(* IEC 61131-3 sources: programs/VI-54/VI-54_20171205/VI-54_20171205/Stations/Screen/LseClass170718/Class/EventJournal (part 2) *)

    // Koordinaten bestimmen
    tmpRoom.xy1.x += to_int(EventConfig.aColumnWidths[3]);
    tmpRoom.xy2.x += to_int(EventConfig.aColumnWidths[3]);

    Graphic.Line( x1      := tmpRoom.xy1.x,
                  y1      := tmpRoom.xy1.y,
                  x2      := tmpRoom.xy2.x,
                  y2      := tmpRoom.xy2.y,
                  attrib  := T_SOLID,
                  color   := sColor);

  end_if;

  //-----------------------------------------------------------------------------------------

END_FUNCTION

FUNCTION VIRTUAL EventJournal::GetEventText
	VAR_INPUT
		pEntry 	: ^_SINGLEALARM;
	END_VAR
	VAR_OUTPUT
		pEventTxt 	: ^_CHAR;
	END_VAR
  VAR
    pText       : ^_CHAR;
    tmpColor    : _COLOR;
    tmpIndex    : UINT;
   	MemVarLabel	: _MEM_VARLABEL;			// pointer to structure to get variables or constants
  END_VAR

  //===============================================================================================
  //  INIT
  //===============================================================================================
  pEventTxt := NIL;

  //===============================================================================================
  //  Übergabeparameter prüfen
  //===============================================================================================
  if (pEntry = NIL) then
    if (IsCon_coSystemLogging = True) then    // KaiAnd
      coSystemLogging.LogEventText("EventJournal::GetEventText(): Übergabeparameter pEntry = NIL" );
    end_if;
    return;
  end_if;

  //===============================================================================================
  //  create the memvarlabel for the defined text
  //===============================================================================================
 	init_MEM_VARLABEL(#MemVarLabel);

  if (pEntry^.ptr <> NIL) then
		// allocate the memory
    if ((Graphic.Memory(#MemVarLabel.ptr, sizeof(_VARLABEL))) <> NIL) then

      MemVarLabel.no := 1;
      MemVarLabel.ptr^.no := 1;
      MemVarLabel.ptr^.info[0].state := POINTER_CHAR;
      MemVarLabel.ptr^.info[0].value := pEntry^.ptr$DINT;
    end_if;
  end_if;

  //===============================================================================================
  //  UNTERSCHEIDUNG DER VERSCHIEDENEN EINTRÄGE
  //===============================================================================================
  case (pEntry^.entrytype) of

      //=======================================================================================
      //  Steuerung wurde eingeschaltet
      //---------------------------------------------------------------------------------------
      EVENT_SWITCHON:

        pEventTxt$^void := NewDoScheme(x0 := EventConfig.SystemOnOff.list,
                                      x1 := EVENT_TEXTSWITCHON,
                                      x2 := EventConfig.SystemOnOff.no);

        if (pEventTxt = NIL) then
          StrNCpy(p0:= #tmpEvTxt[0], x1:=sizeof(_CHAR), p2:="System on", x3:=1, ml:=sizeof(tmpEvTxt)/sizeof(_CHAR));
          pEventTxt := #tmpEvTxt[0];
        end_if;

      //=======================================================================================
      //  Steuerung wurde ausgeschaltet
      //---------------------------------------------------------------------------------------
      EVENT_SWITCHOFF:

        pEventTxt$^void := NewDoScheme(x0 := EventConfig.SystemOnOff.list,
                                      x1 := EVENT_TEXTSWITCHOFF,
                                      x2 := EventConfig.SystemOnOff.no);

        if (pEventTxt = NIL) then
          StrNCpy(p0:= #tmpEvTxt[0], x1:=sizeof(_CHAR), p2:="System off", x3:=1, ml:=sizeof(tmpEvTxt)/sizeof(_CHAR));
          pEventTxt := #tmpEvTxt[0];
        end_if;

      //=======================================================================================
      //  Betriebsart wurde umgeschaltet
      //---------------------------------------------------------------------------------------
      EVENT_OPCHANGE:

        // je nach Betriebsart anderen Text aus Liste holen
        case (pEntry^.para[2]$t_e_OPMode) of
          OPMode_Init:      tmpIndex := EVENT_TEXTOPMODEINIT;
          OPMode_Stop:      tmpIndex := EVENT_TEXTOPMODESTOP;
          OPMode_Setup:     tmpIndex := EVENT_TEXTOPMODESETUP;
          OPMode_Manual:    tmpIndex := EVENT_TEXTOPMODEMANUAL;
          OPMode_SemiAuto:  tmpIndex := EVENT_TEXTOPMODESEMIAUTO;
          OPMode_Automatic: tmpIndex := EVENT_TEXTOPMODEAUTOMATIC;
        else
          if (IsCon_coSystemLogging = True) then    // KaiAnd
            coSystemLogging.LogEventText("EventJournal::GetEventText(): unbekannter Betriebsmodus eingetragen" );
          end_if;
          tmpIndex := EVENT_TEXTOPMODEINIT;
        end_case;

        // Text aus Textliste holen
        pEventTxt$^void := NewDoScheme(x0 := EventConfig.OPMode.list,
                                       x1 := tmpIndex,
                                       x2 := EventConfig.OPMode.no);

        // Prüfen ob Text gefunden wurde
        if (pEventTxt = NIL) then
          StrNCpy(p0:= #tmpEvTxt[0], x1:=sizeof(_CHAR), p2:="change OP mode", x3:=1, ml:=sizeof(tmpEvTxt)/sizeof(_CHAR));
          pEventTxt := #tmpEvTxt[0];
        end_if;

      //=======================================================================================
      //  Login
      //---------------------------------------------------------------------------------------
      EVENT_USERLOGIN:

        pText := StupidTextScheme(Event_TextLogin, EventConfig.LoginLogout.no);
        pText := make_parameterstring(pText, #MemVarLabel, _TRUE);

        // Prüfen ob Text verfügbar
        if (pText = NIL) then
          StrNCpy(p0:= #tmpEvTxt[0], x1:=sizeof(_CHAR), p2:="user login text not found", x3:=1, ml:=sizeof(tmpEvTxt)/sizeof(_CHAR));
        else
          StrNCpy(p0:= #tmpEvTxt[0], x1:=sizeof(_CHAR), p2:=pText, x3:=sizeof(_CHAR), ml:=sizeof(tmpEvTxt)/sizeof(_CHAR));
        end_if;
        pEventTxt := #tmpEvTxt[0];

      //=======================================================================================
      //  Logout
      //---------------------------------------------------------------------------------------
      EVENT_USERLOGOUT:

        // Alarmtext bestimmen
        pText := StupidTextScheme(EVENT_TEXTLOGOUT, EventConfig.LoginLogout.no);
        pText := make_parameterstring(pText, #MemVarLabel, _TRUE);

        // Prüfen ob Text verfügbar
        if (pText = NIL) then
          StrNCpy(p0:= #tmpEvTxt[0], x1:=sizeof(_CHAR), p2:="user logout text not found", x3:=1, ml:=sizeof(tmpEvTxt)/sizeof(_CHAR));
        else
          StrNCpy(p0:= #tmpEvTxt[0], x1:=sizeof(_CHAR), p2:=pText, x3:=sizeof(_CHAR), ml:=sizeof(tmpEvTxt)/sizeof(_CHAR));
        end_if;
        pEventTxt := #tmpEvTxt[0];

      //=======================================================================================
      //  Benutzer-Event
      //---------------------------------------------------------------------------------------
      EVENT_USEREVENT:

        pEventTxt$^void := pEntry^.ptr;

      //=======================================================================================
      //  Datumsänderung
      //---------------------------------------------------------------------------------------
      EVENT_DATECHANGE:

        pEventTxt := GetTextEventDateChange(pEntry);

      //=======================================================================================
      //  Zeitänderung
      //---------------------------------------------------------------------------------------
      EVENT_TIMECHANGE:

        pEventTxt := GetTextEventTimeChange(pEntry);

      //=======================================================================================
      //  Wertänderung
      //---------------------------------------------------------------------------------------
      EVENT_VALUECHANGE:

        pEventTxt := GetTextEventValueChange(pEntry);

      //=======================================================================================
      //  Menüeintrags-Änderung
      //---------------------------------------------------------------------------------------
      EVENT_MENUCHANGE:

        pEventTxt := GetTextEventMenueChange(pEntry);

      //=======================================================================================
      //  Alarm
      //---------------------------------------------------------------------------------------
      EVENT_ALARM :
        // Alarmtext bestimmen
        pEventTxt := create_alarmtext(p0:= pEntry, x1:=false, p2:=#tmpColor);

        // Prüfen ob Text verfügbar
        if (pEventTxt = NIL) then
          if (IsCon_coSystemLogging = True) then    // KaiAnd
            coSystemLogging.LogEventText("EventJournal::GetEventText(): Text für den Alarm nicht gefunden" );
          end_if;
        end_if;

      //=======================================================================================
      //  System Meldungen Kategorie 1
      //---------------------------------------------------------------------------------------
      Event_SystemCat1 :

        // Alarmtext bestimmen
        pText := StupidTextScheme(pEntry^.para[2], EventConfig.SystemEntryCategory1.no);
        pText := make_parameterstring(pText, #MemVarLabel, _TRUE);

        // Prüfen ob Text verfügbar
        if (pText = NIL) then
          StrNCpy(p0:= #tmpEvTxt[0], x1:=sizeof(_CHAR), p2:="system text cat1 not found", x3:=1, ml:=sizeof(tmpEvTxt)/sizeof(_CHAR));
        else
          StrNCpy(p0:= #tmpEvTxt[0], x1:=sizeof(_CHAR), p2:=pText, x3:=sizeof(_CHAR), ml:=sizeof(tmpEvTxt)/sizeof(_CHAR));
        end_if;
        pEventTxt := #tmpEvTxt[0];

      //=======================================================================================
      //  System Meldungen Kategorie 2
      //---------------------------------------------------------------------------------------
      Event_SystemCat2 :

        // Alarmtext bestimmen
        pText := StupidTextScheme(pEntry^.para[2], EventConfig.SystemEntryCategory2.no);
        pText := make_parameterstring(pText, #MemVarLabel, _TRUE);

        // Prüfen ob Text verfügbar
        if (pText = NIL) then
          StrNCpy(p0:= #tmpEvTxt[0], x1:=sizeof(_CHAR), p2:="system text cat2 not found", x3:=1, ml:=sizeof(tmpEvTxt)/sizeof(_CHAR));
        else
          StrNCpy(p0:= #tmpEvTxt[0], x1:=sizeof(_CHAR), p2:=pText, x3:=sizeof(_CHAR), ml:=sizeof(tmpEvTxt)/sizeof(_CHAR));
        end_if;
        pEventTxt := #tmpEvTxt[0];

      //=======================================================================================
      //  System Meldungen Kategorie 3
      //---------------------------------------------------------------------------------------
      Event_SystemCat3 :

        // Alarmtext bestimmen
        pText := StupidTextScheme(pEntry^.para[2], EventConfig.SystemEntryCategory3.no);
        pText := make_parameterstring(pText, #MemVarLabel, _TRUE);

        // Prüfen ob Text verfügbar
        if (pText = NIL) then
          StrNCpy(p0:= #tmpEvTxt[0], x1:=sizeof(_CHAR), p2:="system text cat3 not found", x3:=1, ml:=sizeof(tmpEvTxt)/sizeof(_CHAR));
        else
          StrNCpy(p0:= #tmpEvTxt[0], x1:=sizeof(_CHAR), p2:=pText, x3:=sizeof(_CHAR), ml:=sizeof(tmpEvTxt)/sizeof(_CHAR));
        end_if;
        pEventTxt := #tmpEvTxt[0];

      //=======================================================================================
      //  System Meldungen Kategorie 4
      //---------------------------------------------------------------------------------------
      Event_SystemCat4 :

        // Alarmtext bestimmen
        pText := StupidTextScheme(pEntry^.para[2], EventConfig.SystemEntryCategory4.no);
        pText := make_parameterstring(pText, #MemVarLabel, _TRUE);

        // Prüfen ob Text verfügbar
        if (pText = NIL) then
          StrNCpy(p0:= #tmpEvTxt[0], x1:=sizeof(_CHAR), p2:="system text cat4 not found", x3:=1, ml:=sizeof(tmpEvTxt)/sizeof(_CHAR));
        else
          StrNCpy(p0:= #tmpEvTxt[0], x1:=sizeof(_CHAR), p2:=pText, x3:=sizeof(_CHAR), ml:=sizeof(tmpEvTxt)/sizeof(_CHAR));
        end_if;
        pEventTxt := #tmpEvTxt[0];

      //=======================================================================================
      // Nicht unterstütztes Event
      //---------------------------------------------------------------------------------------
      else
        if (IsCon_coSystemLogging = True) then    // KaiAnd
          coSystemLogging.LogEventText("EventJournal::GetEventText(): Eintrag aus EventJournal nicht unterstützt" );
        end_if;

  end_case;

	// frees the memory
	free_MEM_VARLABEL(#MemVarLabel);

END_FUNCTION

FUNCTION EventJournal::GetEventTime
	VAR_INPUT
		pEntry 	: ^_SINGLEALARM;
		pRetdDate 	: ^DINT;    // V.1.2
		pRetdTime 	: ^DINT;    // V.1.2
	END_VAR
	VAR_OUTPUT
		pString 	: ^_CHAR;
	END_VAR
  VAR
    tmpLength : UDINT;
  	tmpDate   : _DATE;
    tmpTime   : _TIME;
    tmpHlpTxt : ARRAY [0..20] OF _CHAR;
  END_VAR

  // Rückgabewert initialisieren
  pString := NIL;
  if (pRetdDate <> NIL) then     // V.1.2
    pRetdDate^ := 0;
  end_if;
  if (pRetdTime <> NIL) then     // V.1.2
    pRetdTime^ := 0;
  end_if;

  // Übergabeparameter prüfen
  if (pEntry = NIL) then
    if (IsCon_coSystemLogging = True) then    // KaiAnd
      coSystemLogging.LogEventText("EventJournal::GetEventTime(): Übergabeparameter pEntry = NIL");
    end_if;
    return;
  end_if;

  // Datum wandeln
  lasal_to_DATE(p0:=#tmpDate, x1:=pEntry^.date_on);

  // String erzeugen
  format_date(p0:=#tmpHlpTxt[0], p1:=#tmpDate, x2:=SIZE_DDMMYY);

  // String anfügen
  StrCpy(p0:=#tmpEvTxt[0], x1:=sizeof(_CHAR), p2:=#tmpHlpTxt[0], x3:=sizeof(_CHAR));

  // Seperator einfügen
  StrCat(p0:=#tmpEvTxt[0], x1:=sizeof(_CHAR), p2:=" ", x3:=1);

  // Zeit wandeln
  lasal_to_TIME(p0:=#tmpTime, x1:=pEntry^.time_on);

  // String erzeugen
  format_time(p0:=#tmpHlpTxt[0], p1:=#tmpTime, x2:=SIZE_HHMMSS);

  // String anfügen
  StrCat(p0:=#tmpEvTxt[0], x1:=sizeof(_CHAR), p2:=#tmpHlpTxt[0], x3:=sizeof(_CHAR));

  // Länge bestimmen + 0 - Abschluss
  tmpLength := StrLen(txt:=#tmpEvTxt[0], size:=sizeof(_CHAR)) + 1;

  // Pointer auf String zurück liefern
  pString := #tmpEvTxt[0];

  // return also Date and Time as values   V.1.2, KaiAnd
  if (pRetdDate <> NIL) then
    pRetdDate^ := pEntry^.date_on;
  end_if;
  if (pRetdTime <> NIL) then
    pRetdTime^ := pEntry^.time_on;
  end_if;

END_FUNCTION

FUNCTION EventJournal::GetParameter1
	VAR_INPUT
		pEntry 	 : ^_SINGLEALARM;
		pRetDINT : ^DINT;    // V.1.2
	END_VAR
	VAR_OUTPUT
		pString  : ^_CHAR;
	END_VAR
  VAR
    tmpPara1 : DINT;
  END_VAR

  // Rückgabewert initialisieren
  pString  := NIL;
  tmpPara1 := 0;
  if (pRetDINT <> NIL) then     // V.1.2
    pRetDINT^ := 0;
  end_if;

  // Übergabeparameter prüfen
  if (pEntry = NIL) then
    if (IsCon_coSystemLogging = True) then    // KaiAnd
      coSystemLogging.LogEventText("EventJournal::GetParameter1(): Übergabeparameter pEntry = NIL");
    end_if;
    return;
  end_if;

  // Länge prüfen
  #pragma warning(disable:69); // disable warning
  if ( sizeof(tmpEvTxt) < 20 ) then
    if (IsCon_coSystemLogging = True) then    // KaiAnd
      coSystemLogging.LogEventText("EventJournal::GetParameter1(): Länge des Zielstrings zu klein");
    end_if;
    return;
  end_if;
  #pragma warning(default:69);

  //*****************************************************************************
  //** UNTERSCHEIDUNG DER EVENTS                                               **
  //*****************************************************************************

  case pEntry^.entrytype of

    // Alarm
    //*****************************************************************************
    EVENT_ALARM:

      // Prüfen ob Parameter1 verfügbar
      if (pEntry^.no_para >= 1) then
        // Parameter1 steht am letzten Parameter
        tmpPara1 := pEntry^.para[pEntry^.no_para -1];
      else
        if (IsCon_coSystemLogging = True) then    // KaiAnd
          coSystemLogging.LogEventText("EventJournal::GetParameter1(): Kein Parameter1 für Event verfügbar");
        end_if;
      end_if;

    // Alles andere
    //*****************************************************************************
    else

      // Prüfen ob Parameter1 verfügbar
      if (pEntry^.no_para >= 1) then
        // Parameter1 steht immer am ersten Parameter
        tmpPara1 := pEntry^.para[0];
      else
        if (IsCon_coSystemLogging = True) then    // KaiAnd
          coSystemLogging.LogEventText("EventJournal::GetParameter1(): Kein Parameter1 für Event verfügbar");
        end_if;
      end_if;

  end_case;

  // Nummer zu Text wandeln
  DToA(p0:=#tmpEvTxt[0], x1:=tmpPara1, x2:=Event_ConfigParam1, x3:=sizeof(_CHAR));
  pString := #tmpEvTxt[0];

  // return also value     V.1.2, KaiAnd
  if (pRetDINT <> NIL) then
    pRetDINT^ := tmpPara1;
  end_if;

END_FUNCTION

FUNCTION EventJournal::GetAlarmNo
	VAR_INPUT
		pEntry 	 : ^_SINGLEALARM;
		pRetDINT : ^DINT;    // V.1.2
	END_VAR
	VAR_OUTPUT
		pString  : ^_CHAR;
	END_VAR
  VAR
    tmpAlaNo : DINT;
  END_VAR

  // Rückgabewert initialisieren
  pString  := NIL;
  tmpAlaNo := 0;
  if (pRetDINT <> NIL) then     // V.1.2
    pRetDINT^ := 0;
  end_if;

  // Übergabeparameter prüfen
  if (pEntry = NIL) then
    if (IsCon_coSystemLogging = True) then    // KaiAnd
      coSystemLogging.LogEventText("EventJournal::GetAlarmNo(): Übergabeparameter pEntry = NIL");
    end_if;
    return;
  end_if;

  // Länge prüfen
  #pragma warning(disable:69); // disable warning
  if ( sizeof(tmpEvTxt) < 20 ) then
    if (IsCon_coSystemLogging = True) then    // KaiAnd
      coSystemLogging.LogEventText("EventJournal::GetAlarmNo(): Länge des Zielstrings zu klein");
    end_if;
    return;
  end_if;
  #pragma warning(default:69);

  //*****************************************************************************
  //** UNTERSCHEIDUNG DER VERSCHIEDENEN EINTRÄGE                               **
  //*****************************************************************************

  case (pEntry^.entrytype) of

    // Eventeintrag ist ein Alarm bzw. Wertänderung
    //*****************************************************************************
    EVENT_ALARM:

      tmpAlaNo := pEntry^.no;

      // Alarmnummer bzw. Bildnummer zu Text wandeln
      DToA(p0:=#tmpEvTxt[0], x1:=pEntry^.no, x2:=EVENT_CONFIGALARMNO, x3:=sizeof(_CHAR));
      pString := #tmpEvTxt[0];

    // Alles Andere
    //*****************************************************************************
    else

      // es wird keine Zahl dargestellt
      StrCpy(p0:=#tmpEvTxt[0], x1:= sizeof(_CHAR), p2:=" ", x3:=1);
      pString := #tmpEvTxt[0];

  end_case;

  // return also value     V.1.2, KaiAnd
  if (pRetDINT <> NIL) then
    pRetDINT^ := tmpAlaNo;
  end_if;

END_FUNCTION

FUNCTION EventJournal::GetParameter2
	VAR_INPUT
		pEntry 	 : ^_SINGLEALARM;
		pRetDINT : ^DINT;    // V.1.2
	END_VAR
	VAR_OUTPUT
		pString  : ^_CHAR;
	END_VAR
  VAR
    tmpPara2 : DINT;
  END_VAR

  // Rückgabewert initialisieren
  pString  := NIL;
  tmpPara2 := 0;
  if (pRetDINT <> NIL) then     // V.1.2
    pRetDINT^ := 0;
  end_if;

  // Übergabeparameter prüfen
  if (pEntry = NIL) then
    if (IsCon_coSystemLogging = True) then    // KaiAnd
      coSystemLogging.LogEventText("EventJournal::GetParameter2(): Übergabeparameter pEntry = NIL");
    end_if;
    return;
  end_if;

  // Länge prüfen
  #pragma warning(disable:69); // disable warning
  if ( sizeof(tmpEvTxt) < 20 ) then
    if (IsCon_coSystemLogging = True) then    // KaiAnd
      coSystemLogging.LogEventText("EventJournal::GetParameter2(): Länge des Zielstrings zu klein");
    end_if;
    return;
  end_if;
  #pragma warning(default:69);

  //*****************************************************************************
  //** UNTERSCHEIDUNG DER VERSCHIEDENEN EINTRÄGE                               **
  //*****************************************************************************

  case pEntry^.entrytype of

    // Eventeintrag prüfen, ob Parameter2 verfügbar ist
    //*****************************************************************************
    Event_SystemCat1, Event_SystemCat2,
    Event_SystemCat3, Event_SystemCat4,
    Event_UserLogout, Event_UserLogin,
    EVENT_DATECHANGE, EVENT_TIMECHANGE,
    Event_OPChange, Event_MenuChange,
    Event_UserEvent, Event_EventEntry,
    Event_ValueChange:

      tmpPara2 := pEntry^.para[1];

      // Parameter2 zu Text wandeln
      DToA(p0:=#tmpEvTxt[0], x1:=pEntry^.para[1], x2:=EVENT_CONFIGPARAM2, x3:=sizeof(_CHAR));
      pString := #tmpEvTxt[0];

    // Alles Andere
    //*****************************************************************************
    else

      // es wird keine Zahl dargestellt
      StrCpy(p0:=#tmpEvTxt[0], x1:= sizeof(_CHAR), p2:=" ", x3:=1);
      pString := #tmpEvTxt[0];

  end_case;

  // return also value     V.1.2, KaiAnd
  if (pRetDINT <> NIL) then
    pRetDINT^ := tmpPara2;
  end_if;

END_FUNCTION

FUNCTION EventJournal::GetTextEventDateChange
	VAR_INPUT
		pEntry 	: ^_SINGLEALARM;
	END_VAR
	VAR_OUTPUT
		pString 	: ^_CHAR;
	END_VAR
  VAR
    pText       : ^_CHAR;
    tmpLength   : UDINT;
    tmpHlpTxt   : ARRAY[0..49] OF _CHAR;
    tmpVariable : _VARIABLE;
    tmpDate     : _DATE;
    szValueTxt  : ARRAY[0..199] of _CHAR;
  END_VAR

  // Variableninformation vom Server holen
  if (VarList_GetSingleVariable(p0:=#tmpVariable, x1:=to_udint(pEntry^.para[2])) = true) then

    // Variablentext holen
    //*****************************************************************************
    pText := VarList_GetTextByNo(x0:=to_udint(pEntry^.para[2]), x1:=0);

    // Prüfen ob UnitText verfügbar
    if (pText <> NIL) then
      // String auf Ziel kopieren
      StrNCpy(p0:=#tmpEvTxt[0], x1:=sizeof(_CHAR), p2:=pText, x3:=sizeof(_CHAR), ml:=sizeof(tmpEvTxt)/sizeof(_CHAR));
    else
      // String auf Ziel kopieren
      StrNCpy(p0:=#tmpEvTxt[0], x1:=sizeof(_CHAR), p2:="no text defined", x3:=1, ml:=sizeof(tmpEvTxt)/sizeof(_CHAR));
    end_if;

    tmpLength := StrSize(p0:=#tmpEvTxt[0], x1:=sizeof(_CHAR));

    //*****************************************************************************
    // Wertänderung zusammenbauen
    //*****************************************************************************

    // Alten Wert wandeln
    lasal_to_DATE(p0:=#tmpDate, x1:=pEntry^.para[3]);
    format_date(#tmpHlpTxt[0], #tmpDate, SIZE_DDMMYYYY);

    StrCpy(p0:=#szValueTxt[0], x1:=sizeof(_CHAR), p2:=": ", x3:=1);

    StrCat(p0:=#szValueTxt[0] ,x1:=sizeof(_CHAR), p2 := #tmpHlpTxt[0], x3:=sizeof(_CHAR));

    // Neuen Wert wandeln
    lasal_to_DATE(p0:=#tmpDate, x1:=pEntry^.para[4]);
    format_date(#tmpHlpTxt[0], #tmpDate, SIZE_DDMMYYYY);

    StrCat(p0:=#szValueTxt[0], x1:=sizeof(_CHAR), p2:= " -> ", x3 := 1);
    StrCat(p0:=#szValueTxt[0], x1:=sizeof(_CHAR), p2:= #tmpHlpTxt[0], x3 := sizeof(_CHAR));

    tmpLength += StrSize(p0:=#szValueTxt[0], x1:=sizeof(szValueTxt[0])) + sizeof(szValueTxt[0]);

    if (tmpLength <= sizeof(tmpEvTxt)) then
      StrCat(p0:=#tmpEvTxt[0], x1:=sizeof(_CHAR), p2:=#szValueTxt[0], x3:=sizeof(_CHAR));
    else
      StrCpy(p0:=#tmpEvTxt[0], x1:=sizeof(_CHAR), p2:="text too long", x3:=1);
    end_if;

  else
      StrCpy(p0:=#tmpEvTxt[0], x1:=sizeof(_CHAR), p2:="no variable defined", x3:=1);
  end_if;

  // Pointer mit Ergebnis zurück liefern
  pString := #tmpEvTxt[0];

END_FUNCTION

FUNCTION EventJournal::GetTextEventTimeChange
	VAR_INPUT
		pEntry 	: ^_SINGLEALARM;
	END_VAR
	VAR_OUTPUT
		pString 	: ^_CHAR;
	END_VAR
  VAR
    pText       : ^_CHAR;
    tmpLength   : UDINT;
    tmpHlpTxt   : ARRAY[0..49] OF _CHAR;
    tmpVariable : _VARIABLE;
    tmpTime     : _TIME;
    szValueTxt  : ARRAY[0..199] of _CHAR;
  END_VAR

  // Variableninformation vom Server holen
  if (VarList_GetSingleVariable(p0:=#tmpVariable, x1:=to_udint(pEntry^.para[2])) = true) then

    // Variablentext holen
    //*****************************************************************************
    pText := VarList_GetTextByNo(x0:=to_udint(pEntry^.para[2]), x1:=0);

    // Prüfen ob UnitText verfügbar
    if (pText <> NIL) then
      // String auf Ziel kopieren
      StrNCpy(p0:=#tmpEvTxt[0], x1:=sizeof(_CHAR), p2:=pText, x3:=sizeof(_CHAR), ml:=sizeof(tmpEvTxt)/sizeof(_CHAR));
    else
      // String auf Ziel kopieren
      StrNCpy(p0:=#tmpEvTxt[0], x1:=sizeof(_CHAR), p2:="no text defined", x3:=1, ml:=sizeof(tmpEvTxt)/sizeof(_CHAR));
    end_if;

    tmpLength := StrSize(p0:=#tmpEvTxt[0], x1:=sizeof(_CHAR));

    //*****************************************************************************
    // Wertänderung zusammenbauen
    //*****************************************************************************

    // alten Wert wandeln
    lasal_to_TIME(p0:=#tmpTime, x1:=pEntry^.para[3]);
    format_time(#tmpHlpTxt[0], #tmptime, SIZE_HHMMSS);

    StrCpy(p0:=#szValueTxt[0], x1:=sizeof(_CHAR), p2:=": ", x3:=1);

    StrCat(p0:=#szValueTxt[0] ,x1:=sizeof(_CHAR), p2:=#tmpHlpTxt[0], x3:=sizeof(_CHAR));

    // neuen Wert wandeln
    lasal_to_TIME(p0:=#tmpTime, x1:=pEntry^.para[4]);
    format_time(#tmpHlpTxt[0], #tmpTime, SIZE_HHMMSS);

    StrCat(p0:= #szValueTxt[0], x1:=sizeof(_CHAR), p2:=" -> ", x3:=1);
    StrCat(p0:= #szValueTxt[0], x1:=sizeof(_CHAR), p2:=#tmpHlpTxt[0], x3:=sizeof(_CHAR));

    tmpLength += StrSize(p0:=#szValueTxt[0], x1:=sizeof(szValueTxt[0])) + sizeof(szValueTxt[0]);

    if (tmpLength <= sizeof(tmpEvTxt)) then
      StrCat(p0:=#tmpEvTxt[0], x1:=sizeof(_CHAR), p2:=#szValueTxt[0], x3:=sizeof(_CHAR));
    else
      StrCpy(p0:=#tmpEvTxt[0], x1:=sizeof(_CHAR), p2:="text too long", x3:=1);
    end_if;

  else
      StrCpy(p0:=#tmpEvTxt[0], x1:=sizeof(_CHAR), p2:="no variable defined", x3:=1);
  end_if;

  // Pointer mit Ergebnis zurück liefern
  pString := #tmpEvTxt[0];

END_FUNCTION

FUNCTION EventJournal::GetTextEventValueChange
	VAR_INPUT
		pEntry 	: ^_SINGLEALARM;
	END_VAR
	VAR_OUTPUT
		pString 	: ^_CHAR;
	END_VAR
  VAR
    pText       : ^_CHAR;
    tmpLength   : UDINT;
    tmpResult   : _RESULT;
    tmpHlpTxt   : ARRAY[0..49] OF _CHAR;
    tmpVariable : _VARIABLE;
    szValueTxt  : ARRAY[0..199] of _CHAR;
    szUnitTxt   : ARRAY[0..49] of _CHAR;
  END_VAR

  // Variableninformation vom Server holen
  if (VarList_GetSingleVariable(p0:=#tmpVariable, x1:=to_udint(pEntry^.para[2])) = true) then

    // Variablentext holen
    //*****************************************************************************
    pText := VarList_GetTextByNo(x0:=to_udint(pEntry^.para[2]), x1:=0);

    // Prüfen ob UnitText verfügbar
    if (pText <> NIL) then
      // String auf Ziel kopieren
      StrNCpy(p0:=#tmpEvTxt[0], x1:=sizeof(_CHAR), p2:=pText, x3:=sizeof(_CHAR), ml:=sizeof(tmpEvTxt)/sizeof(_CHAR));
    else
      // String auf Ziel kopieren
      StrNCpy(p0:=#tmpEvTxt[0], x1:=sizeof(_CHAR), p2:="no text defined", x3:=1, ml:=sizeof(tmpEvTxt)/sizeof(_CHAR));
    end_if;

    tmpLength := StrSize(p0:=#tmpEvTxt[0], x1:=sizeof(_CHAR));

    //*****************************************************************************
    // Wertänderung zusammenbauen
    //*****************************************************************************

    //Unit holen
    pText := VarList_GetTextByNo(x0:=to_udint(pEntry^.para[2]), x1:=5);
    if (pText = NIL)  then  // KaiAnd: unit is fine but not needed!!

      StrCpy(p0:=#szUnitTxt[0], x1:=sizeof(_CHAR), p2:=" [ ] ", x3:=1);

    else

      // [ einfügen
      StrCpy(p0:=#szUnitTxt[0], x1:=sizeof(_CHAR), p2:=" [", x3:=1);
      // String mit Unit-Text kopieren
      StrCat(p0:=#szUnitTxt[0], x1:=sizeof(_CHAR), p2:=pText, x3:=sizeof(_CHAR));
      // ] einfügen
      StrCat(p0:=#szUnitTxt[0], x1:=sizeof(_CHAR), p2:="] ", x3:=1);

    end_if;

    // Alten Wert wandeln
    tmpResult.ftype := RES_NUMERIC;
    tmpResult.value := pEntry^.para[3];

    // Wert mit eingestellter Einheit umrechnen
    recalculate(p0:=#tmpResult, p1:=#tmpVariable, x2:=TRUE);

    // Wert mit eingestellter Unit formatieren
    format_value(p0:=#tmpHlpTxt[0], x1:=tmpResult.value, p2:=#tmpVariable.info, p3:=NIL);

    StrCpy(p0:=#szValueTxt[0], x1:=sizeof(_CHAR), p2:=": ", x3:=1);
    StrCat(p0:=#szValueTxt[0], x1:=sizeof(_CHAR), p2:=#tmpHlpTxt[0], x3:=sizeof(_CHAR));
    StrCat(p0:=#szValueTxt[0], x1:=sizeof(_CHAR), p2:=#szUnitTxt[0], x3:= sizeof(_CHAR));

    // Neuen Wert wandeln
    tmpResult.value := pEntry^.para[4];

    // Wert mit eingestellter Einheit umrechnen
    recalculate(p0:=#tmpResult, p1:=#tmpVariable, x2:=TRUE);

    // Wert mit eingestellter Unit formatieren
    format_value(p0:=#tmpHlpTxt[0], x1:=tmpResult.value, p2:=#tmpVariable.info, p3:=NIL);

    StrCat(p0:=#szValueTxt[0], x1:=sizeof(_CHAR), p2:=" -> ", x3:=1);
    StrCat(p0:=#szValueTxt[0], x1:=sizeof(_CHAR), p2:=#tmpHlpTxt[0], x3:=sizeof(_CHAR));
    StrCat(p0:=#szValueTxt[0], x1:=sizeof(_CHAR), p2:=#szUnitTxt[0], x3:=sizeof(_CHAR));

    tmpLength += StrSize(p0:=#szValueTxt[0], x1:=sizeof(szValueTxt[0])) + sizeof(szValueTxt[0]);

    if (tmpLength <= sizeof(tmpEvTxt)) then
      StrCat(p0:=#tmpEvTxt[0], x1:=sizeof(_CHAR), p2:=#szValueTxt[0], x3:=sizeof(_CHAR));
    else
      StrCpy(p0:=#tmpEvTxt[0], x1:=sizeof(_CHAR), p2:="text too long", x3:=1);
    end_if;

  else
      StrCpy(p0:=#tmpEvTxt[0], x1:=sizeof(_CHAR), p2:="no variable defined", x3:=1);
  end_if;

  // Pointer mit Ergebnis zurück liefern
  pString := #tmpEvTxt[0];

END_FUNCTION

FUNCTION EventJournal::GetTextEventMenueChange
	VAR_INPUT
		pEntry 	: ^_SINGLEALARM;
	END_VAR
	VAR_OUTPUT
		pString 	: ^_CHAR;
	END_VAR
  VAR
    pText       : ^_CHAR;
    tmpLength   : UDINT;
    tmpVariable : _VARIABLE;
    szValueTxt  : ARRAY[0..199] of _CHAR;
    pMenue      : ^_LSEMENU;
    pLine       : ^_LINEINFO;
    pMenuText   : ^void;
  END_VAR

  // Variableninformation vom Server holen
  if (VarList_GetSingleVariable(p0:=#tmpVariable, x1:=to_udint(pEntry^.para[2])) = true) then

    // Variablentext holen
    //*****************************************************************************
    pText := VarList_GetTextByNo(x0:=to_udint(pEntry^.para[2]), x1:=0);

    // Prüfen ob UnitText verfügbar
    if (pText <> NIL) then
      // String auf Ziel kopieren
      StrNCpy(p0:=#tmpEvTxt[0], x1:=sizeof(_CHAR), p2:=pText, x3:=sizeof(_CHAR), ml:=sizeof(tmpEvTxt)/sizeof(_CHAR));
    else
      // String auf Ziel kopieren
      StrNCpy(p0:=#tmpEvTxt[0], x1:=sizeof(_CHAR), p2:="no text defined", x3:=1, ml:=sizeof(tmpEvTxt)/sizeof(_CHAR));
    end_if;

    tmpLength := StrSize(p0:=#tmpEvTxt[0], x1:=sizeof(_CHAR));

    //*****************************************************************************
    // Wertänderung zusammenbauen
    //*****************************************************************************

    // Zeiger auf Menü holen
    pMenue := get_LSEMENU(pEntry^.para[5]$UDINT);

    if (pMenue <> NIL) then

      // Alten Wert wandeln
      // Zeiger auf erste Menüzeile holen
      pLine := pMenue^.mem_lineinfo.ptr;

      if (pLine <> NIL) then

        // Zeiger auf gewünschte Zeilennummer bilden
        pLine += pEntry^.para[3] * sizeof(_LINEINFO);

        // Zeiger auf Menü-Text holen
        pMenuText := get_ANYTHING(#pLine^.anypara.anything, NIL);

        if (pMenuText <> NIL) then

          StrCpy(p0:=#szValueTxt[0], x1:=sizeof(_CHAR), p2:=": ", x3:=1);
          StrCat(p0:=#szValueTxt[0] ,x1:=sizeof(_CHAR), p2:=pMenuText, x3:=sizeof(_CHAR));

          // Neuen Wert wandeln
          // Zeiger auf gewünschte Zeilennummer bilden
          pLine -= pEntry^.para[3] * sizeof(_LINEINFO);
          pLine += pEntry^.para[4] * sizeof(_LINEINFO);

          // Zeiger auf Menü-Text holen
          pMenuText := get_ANYTHING(#pLine^.anypara.anything, NIL);

          StrCat(p0:= #szValueTxt[0] ,x1:=sizeof(_CHAR), p2:=" -> ", x3 := 1);
          StrCat(p0:= #szValueTxt[0] ,x1:=sizeof(_CHAR), p2:=pMenuText, x3 := sizeof(_CHAR));

          tmpLength += StrSize(p0:=#szValueTxt[0], x1:=sizeof(szValueTxt[0])) + sizeof(szValueTxt[0]);

          if (tmpLength <= sizeof(tmpEvTxt)) then
            StrCat(p0:=#tmpEvTxt[0], x1:=sizeof(_CHAR), p2:=#szValueTxt[0], x3:=sizeof(_CHAR));
          end_if;

        else
          StrCpy(p0:=#tmpEvTxt[0], x1:=sizeof(_CHAR), p2:="no variable defined", x3:=1);
        end_if;

      else
        StrCpy(p0:=#tmpEvTxt[0], x1:=sizeof(_CHAR), p2:="no variable defined", x3:=1);
      end_if;

    else
      StrCpy(p0:=#tmpEvTxt[0], x1:=sizeof(_CHAR), p2:="no variable defined", x3:=1);
    end_if;

    if (tmpLength <= sizeof(tmpEvTxt)) then
      StrCat(p0:=#tmpEvTxt[0], x1:=sizeof(_CHAR), p2:=#szValueTxt[0], x3:=sizeof(_CHAR));
    end_if;

  else
      StrCpy(p0:=#tmpEvTxt[0], x1:=sizeof(_CHAR), p2:="no variable defined", x3:=1);
  end_if;

  // Pointer mit Ergebnis zurück liefern
  pString := #tmpEvTxt[0];

END_FUNCTION

FUNCTION EventJournal::GetTheUrgeValues
	VAR_INPUT
		pio 	: ^_IO;
	END_VAR
	VAR_OUTPUT
		bSuccessful 	: BOOL;
	END_VAR
  VAR
    tmpCounter  : USINT;
    tmpResult   : _RESULT;
    tmpVariable : _VARIABLE;
    tmpVarLabel : _VARLABEL;
  END_VAR

  bSuccessful := true;

  // loop to check all variables
  for tmpCounter := 0 to sizeof(aVarSingle) / sizeof(aVarSingle[0]) - 1 do

    // check if variable is a dataserver
    if (aVarSingle[tmpCounter].state = VAR_VAL) then

      // build varlabel
      tmpVarLabel.no      := 1;
      tmpVarLabel.info[0] := aVarSingle[tmpCounter];

      // get server-value
      if VarList_GetSystemData( p0 := #tmpResult,
                                p1 := #tmpVariable,
                                p2 := #tmpVarLabel,
                                x3 := false) = true then

        // save the new value + change checksum
        EventConfig.aColumnWidths[tmpCounter] := tmpResult.value;

      else
        bSuccessful := false;
      end_if;

    end_if;

  end_for;

END_FUNCTION

FUNCTION EventJournal::GetTheUrge
	VAR_INPUT
		pio 	: ^_IO;
	END_VAR
	VAR_OUTPUT
		bSuccessful 	: BOOL;
	END_VAR
  VAR
    tmpCounter      : USINT;
	  pVarLabel       : ^_VARLABEL;
    pColor          : ^_COLOR;
    pHelpAnyThing   : ^_ANYTHING;
    tmpIndex        : UINT;
    tmpCount        : UINT;
    tmpColType      : UINT;
  END_VAR

  // Gültiger Übergabeparameter?
  if (pio <> NIL) & (pio^.theurge <> NIL) then

    // Richtige Version des UDCs?
    if (pio^.theurge^.info = Event_UDCVersion) then

      bSuccessful := true;

      // variable informations
      //--------------------------------------------------------------
      // check number of variables
      if (pio^.theurge^.memvarlabel.no = Event_VariableNo) then

        // pointer to variable informations
        pVarLabel := pio^.theurge^.memvarlabel.ptr;

        // loop to store all parameter
        for tmpCounter:=0 to (sizeof(aVarSingle)/sizeof(aVarSingle[0]) -1) do

          // save variable informations
          aVarSingle[tmpCounter] := pVarLabel^.info[0];

          // check for constant
          if (aVarSingle[tmpCounter].state = CONST_VAL) then
            EventConfig.aColumnWidths[tmpCounter] := aVarSingle[tmpCounter].value;
          end_if;

          // step to next variable
          pVarLabel += sizeof(_VARLABEL);

        end_for;

      else
        bSuccessful := false;
      end_if;

      // Index des Textschemas holen
      //-----------------------------------------------------------------------------------------
      if (pio^.theurge^.memanything.no = Event_TextschemeNo) then

        pHelpAnyThing := pio^.theurge^.memanything.ptr;

        // Schema ein Textschema?
        if (pHelpAnyThing^.list = TEXTSCHEME) then
          EventConfig.SystemOnOff.list := pHelpAnyThing^.list;
          EventConfig.SystemOnOff.no   := pHelpAnyThing^.no;
        else
          EventConfig.SystemOnOff.list := DEFLST;
          EventConfig.SystemOnOff.no   := DEFSCOPE;
          if (IsCon_coSystemLogging = True) then    // KaiAnd
            coSystemLogging.LogEventText("EventJournal::GetTheUrge(): Verweis auf Textliste konnte nicht bestimmt werden");
          end_if;
        end_if;

        pHelpAnyThing += sizeof(_ANYTHING);

        // Schema ein Textschema?
        if (pHelpAnyThing^.list = TEXTSCHEME) then
          EventConfig.OPMode.list := pHelpAnyThing^.list;
          EventConfig.OPMode.no   := pHelpAnyThing^.no;
        else
          EventConfig.OPMode.list := DEFLST;
          EventConfig.OPMode.no   := DEFSCOPE;
          if (IsCon_coSystemLogging = True) then    // KaiAnd
            coSystemLogging.LogEventText("EventJournal::GetTheUrge(): Verweis auf Textliste konnte nicht bestimmt werden");
          end_if;
        end_if;

        pHelpAnyThing += sizeof(_ANYTHING);

        // Schema ein Textschema?
        if (pHelpAnyThing^.list = TEXTSCHEME) then
          EventConfig.LoginLogout.list := pHelpAnyThing^.list;
          EventConfig.LoginLogout.no   := pHelpAnyThing^.no;
        else
          EventConfig.LoginLogout.list := DEFLST;
          EventConfig.LoginLogout.no   := DEFSCOPE;
          if (IsCon_coSystemLogging = True) then    // KaiAnd
            coSystemLogging.LogEventText("EventJournal::GetTheUrge(): Verweis auf Textliste konnte nicht bestimmt werden");
          end_if;
        end_if;

        pHelpAnyThing += sizeof(_ANYTHING);

        // Schema ein Textschema?
        if (pHelpAnyThing^.list = TEXTSCHEME) then
          EventConfig.SystemEntryCategory1.list := pHelpAnyThing^.list;
          EventConfig.SystemEntryCategory1.no   := pHelpAnyThing^.no;
        else
          EventConfig.SystemEntryCategory1.list := DEFLST;
          EventConfig.SystemEntryCategory1.no   := DEFSCOPE;
          if (IsCon_coSystemLogging = True) then    // KaiAnd
            coSystemLogging.LogEventText("EventJournal::GetTheUrge(): Verweis auf Textliste konnte nicht bestimmt werden");
          end_if;
        end_if;

        pHelpAnyThing += sizeof(_ANYTHING);

        // Schema ein Textschema?
        if (pHelpAnyThing^.list = TEXTSCHEME) then
          EventConfig.SystemEntryCategory2.list := pHelpAnyThing^.list;
          EventConfig.SystemEntryCategory2.no   := pHelpAnyThing^.no;
        else
          EventConfig.SystemEntryCategory2.list := DEFLST;
          EventConfig.SystemEntryCategory2.no   := DEFSCOPE;
          if (IsCon_coSystemLogging = True) then    // KaiAnd
            coSystemLogging.LogEventText("EventJournal::GetTheUrge(): Verweis auf Textliste konnte nicht bestimmt werden" );
          end_if;
        end_if;

        pHelpAnyThing += sizeof(_ANYTHING);

        // Schema ein Textschema?
        if (pHelpAnyThing^.list = TEXTSCHEME) then
          EventConfig.SystemEntryCategory3.list := pHelpAnyThing^.list;
          EventConfig.SystemEntryCategory3.no   := pHelpAnyThing^.no;
        else
          EventConfig.SystemEntryCategory3.list := DEFLST;
          EventConfig.SystemEntryCategory3.no   := DEFSCOPE;
          if (IsCon_coSystemLogging = True) then    // KaiAnd
            coSystemLogging.LogEventText("EventJournal::GetTheUrge(): Verweis auf Textliste konnte nicht bestimmt werden" );
          end_if;
        end_if;

        pHelpAnyThing += sizeof(_ANYTHING);

        // Schema ein Textschema?
        if (pHelpAnyThing^.list = TEXTSCHEME) then
          EventConfig.SystemEntryCategory4.list := pHelpAnyThing^.list;
          EventConfig.SystemEntryCategory4.no   := pHelpAnyThing^.no;
        else
          EventConfig.SystemEntryCategory4.list := DEFLST;
          EventConfig.SystemEntryCategory4.no   := DEFSCOPE;
          if (IsCon_coSystemLogging = True) then    // KaiAnd
            coSystemLogging.LogEventText("EventJournal::GetTheUrge(): Verweis auf Textliste konnte nicht bestimmt werden" );
          end_if;
        end_if;

        pHelpAnyThing += sizeof(_ANYTHING);

      else
        bSuccessful := false;
      end_if;

      // color informations
      //--------------------------------------------------------------
      // check number of colors
      tmpCount := 0;
      if (pio^.theurge^.memcolor.no = Event_ColorNo) then

        // pointer to color informations
        pColor := pio^.theurge^.memcolor.ptr;

        while (tmpCount < pio^.theurge^.memcolor.no) do

          // Jede Kategorie hat 2 Farben
          tmpIndex   := tmpCount / 2;
          // Typ der Farbe (BgColor und TxtColor abwechseln im UDC eingetragen)
          tmpColType := tmpCount MOD 2;

          // Textfarbe oder Hintergrundfarbe
          case (tmpColType) of

            0:
                EventConfig.aCategorieColors[tmpIndex].Cat_TextColor := pColor^;

            1:
                EventConfig.aCategorieColors[tmpIndex].Cat_BgColor   := pColor^;

          end_case;

          pColor   += sizeof(_COLOR);
          tmpCount += 1;
        end_while;

      else
        bSuccessful := false;
      end_if;

    else
      bSuccessful := false;
      if (IsCon_coSystemLogging = True) then    // KaiAnd
        coSystemLogging.LogEventText("EventJournal::GetTheUrge(): Falsche Version des UDCs");
      end_if;
    end_if;

  else
    bSuccessful := false;
    if (IsCon_coSystemLogging = True) then    // KaiAnd
      coSystemLogging.LogEventText("EventJournal::GetTheUrge(): Ungültiger Übergabeparameter");
    end_if;
  end_if;

END_FUNCTION

FUNCTION EventJournal::WriteEventTime
	VAR_INPUT
		pEntry 	: ^_SINGLEALARM;
		pRoom 	: ^_ROOM;
		sFont 	: _FONT;
		sTextColor 	: _COLOR;
		sBackColor 	: _COLOR;
	END_VAR
	VAR_OUTPUT
		bSuccessful : BOOL;
	END_VAR
  VAR
    pString    : ^_CHAR;
  END_VAR

  // Übergabeparameter prüfen
  if ((pEntry = NIL) | (pRoom = NIL) )then
    bSuccessful := false;
    return;
  else
    bSuccessful := true;
  end_if;

  // Text bestimmen
  pString := GetEventTime(pEntry:=pEntry, pRetdDate:=NIL, pRetdTime:=NIL);

  // Wenn kein Text verfügbar ist
  if (pString = NIL) then
    StrCpy(p0:= #tmpEvTxt[0], x1:=sizeof(_CHAR), p2:="01.01.70  00:00", x3:=1);
    pString := #tmpEvTxt[0];
  end_if;

  // Text ausgeben
  OutTextAlign( p0 := pString,
                x1 := 0,
                p1 := pRoom,
                x2 := sFont,
                x3 := EVENT_ATTRSTANDARD OR EVENT_ATTRTIME,
                x9 := _DEFFRAME,
                x4 := sTextColor,
                x5 := sBackColor,
                x6 := sBackColor,
                x7 := sizeof(pString^));

END_FUNCTION

FUNCTION EventJournal::WriteParameter1
	VAR_INPUT
		pEntry 	: ^_SINGLEALARM;
		pRoom 	: ^_ROOM;
		sFont 	: _FONT;
		sTextColor 	: _COLOR;
		sBackColor 	: _COLOR;
	END_VAR
	VAR_OUTPUT
		bSuccessful : BOOL;
	END_VAR
  VAR
    pString     : ^_CHAR;
  END_VAR

  // Übergabeparameter prüfen
  if ((pEntry = NIL) | (pRoom = NIL)) then
    bSuccessful := false;
    return;
  else
    bSuccessful := true;
  end_if;

  // Text bestimmen
  pString := GetParameter1(pEntry:=pEntry, pRetDINT:=NIL);

  // Wenn kein Text verfügbar ist
  if (pString = NIL) then
    StrCpy(p0:=#tmpEvTxt[0], x1:=sizeof(_CHAR), p2:= "------", x3:=1);
    pString := #tmpEvTxt[0];
  end_if;

  // Text ausgeben
  OutTextAlign( p0 := pString,
                x1 := 0,
                p1 := pRoom,
                x2 := sFont,
                x3 := EVENT_ATTRSTANDARD OR Event_AttrParam1,
                x9 := _DEFFRAME,
                x4 := sTextColor,
                x5 := sBackColor,
                x6 := sBackColor,
                x7 := sizeof(pString^));

END_FUNCTION

FUNCTION EventJournal::WriteAlarmNo
	VAR_INPUT
		pEntry 	: ^_SINGLEALARM;
		pRoom 	: ^_ROOM;
		sFont 	: _FONT;
		sTextColor 	: _COLOR;
		sBackColor 	: _COLOR;
	END_VAR
	VAR_OUTPUT
		bSuccessful : BOOL;
	END_VAR
  VAR
    pString     : ^_CHAR;
  END_VAR

  // Übergabeparameter prüfen
  if ((pEntry = NIL) | (pRoom = NIL)) then
    bSuccessful := false;
    return;
  else
    bSuccessful := true;
  end_if;

  // Text bestimmen
  pString := GetAlarmNo(pEntry:=pEntry, pRetDINT:=NIL);

  // Prüfen ob Text verfügbar ist
  if (pString <> NIL) then

    // Text ausgeben
    OutTextAlign( p0 := pString,
                  x1 := 0,
                  p1 := pRoom,
                  x2 := sFont,
                  x3 := EVENT_ATTRSTANDARD OR EVENT_ATTRALARMNO,
                  x9 := _DEFFRAME,
                  x4 := sTextColor,
                  x5 := sBackColor,
                  x6 := sBackColor,
                  x7 := sizeof(pString^));
  end_if;

END_FUNCTION

FUNCTION EventJournal::WriteParameter2
	VAR_INPUT
		pEntry 	: ^_SINGLEALARM;
		pRoom 	: ^_ROOM;
		sFont 	: _FONT;
		sTextColor 	: _COLOR;
		sBackColor 	: _COLOR;
	END_VAR
	VAR_OUTPUT
		bSuccessful	: BOOL;
	END_VAR
  VAR
    pString     : ^_CHAR;
  END_VAR

  // Übergabeparameter prüfen
  if ((pEntry = NIL) | (pRoom = NIL)) then
    bSuccessful := false;
    return;
  else
    bSuccessful := true;
  end_if;

  // Text bestimmen
  pString := GetParameter2(pEntry:=pEntry, pRetDINT:=NIL);

  // Prüfen ob Text verfügbar ist
  if (pString <> NIL) then

    // Text ausgeben
    OutTextAlign( p0 := pString,
                  x1 := 0,
                  p1 := pRoom,
                  x2 := sFont,
                  x3 := EVENT_ATTRSTANDARD OR EVENT_ATTRPARAM2,
                  x9 := _DEFFRAME,
                  x4 := sTextColor,
                  x5 := sBackColor,
                  x6 := sBackColor,
                  x7 := sizeof(pString^));
  end_if;

END_FUNCTION

FUNCTION EventJournal::WriteEventText
	VAR_INPUT
		pEntry 	: ^_SINGLEALARM;
		pRoom 	: ^_ROOM;
		sFont 	: _FONT;
		sTextColor 	: _COLOR;
		sBackColor 	: _COLOR;
	END_VAR
	VAR_OUTPUT
		bSuccessful : BOOL;
	END_VAR
  VAR
    pString     : ^_CHAR;
    tmpTest     :  DINT;
  END_VAR

  // Übergabeparameter prüfen
  //-----------------------------------------------------------------------------------------
  if ((pEntry = NIL) | (pRoom = NIL)) then
    bSuccessful := false;
    return;
  else
    bSuccessful := true;
  end_if;

  tmpTest := 1989;

  // Text besorgen
  pString := GetEventText(pEntry:=pEntry);

  if (tmpTest <> 1989) then
    TRACE_ERR("Achtung: Speicherschreiber am Stack");
    (0)$^DINT^ := 0;
  end_if;

  // Prüfen ob Text verfügbar ist
  if (pString = NIL) then

    // Infotext bauen, wenn kein Text verfügbar ist
    StrNCpy(p0 := #tmpText[0],
            x1 := sizeof(_CHAR),
            p2 := " TEXT IS NOT DEFINED IN LSE",
            x3 := 1, // HubChr hardcoded source string is always ascii
            ml := sizeof(tmpText)/sizeof(_CHAR));

    pString := #tmpText[0];

  else
    // shift text in order to put a BLANK in front of the text  HubChr
    StrNCpy(p0 := #tmpText[1],
            x1 := sizeof(_CHAR),
            p2 := pString,
            x3 := sizeof(_CHAR),
            ml := sizeof(tmpText)/sizeof(_CHAR));
    tmpText[0] := ' '; // put BLANK in first character

    pString := #tmpText[0];

  end_if;

  // Text ausgeben
  OutTextAlign(p0 := pString,
               x1 := 0,
               p1 := pRoom,
               x2 := sFont,
               x3 := EVENT_ATTRSTANDARD OR EVENT_ATTRTEXT,
               x9 := _DEFFRAME,
               x4 := sTextColor,
               x5 := sBackColor,
               x6 := sBackColor,
               x7 := sizeof(pString^));

END_FUNCTION

FUNCTION EventJournal::WriteEventEntry
	VAR_INPUT
		pEntry 	: ^_SINGLEALARM;
		pRoom 	: ^_ROOM;
		sFont 	: _FONT;
		sTextColor 	: _COLOR;
		sBackColor 	: _COLOR;
	END_VAR
	VAR_OUTPUT
		bSuccessful : BOOL;
	END_VAR
  VAR
  	tmpRoom    : _ROOM;
  END_VAR

  // Übergabeparameter prüfen
  if ((pEntry = NIL) | (pRoom = NIL)) then
    bSuccessful := false;
    return;
  else
    bSuccessful := true;
  end_if;

  // Leere Zeile ausgeben mit den richtigen Farben falls zuwenig Spalten für die gesamte Breite definiert sind
  Graphic.Beam(x1:=pRoom^.xy1.x, y1:=pRoom^.xy1.y, x2:=pRoom^.xy2.x, y2:=pRoom^.xy2.y, attrib:=EVENT_ATTRSTANDARD  , color:= sBackColor);

  // Platz definieren
  tmpRoom.xy1.x := pRoom^.xy1.x;
  tmpRoom.xy1.y := pRoom^.xy1.y;
  tmpRoom.xy2.x := pRoom^.xy1.x;
  tmpRoom.xy2.y := pRoom^.xy2.y;

  // Eventzeit schreiben
  //------------------------------------------------------------
  // Prüfen ob Zeit dargestellt werden soll
  if (ColumnChoice AND 2#00001) then

    // Platz für Eventzeit bestimmen
    tmpRoom.xy1.x := tmpRoom.xy1.x;
    tmpRoom.xy2.x := tmpRoom.xy1.x + to_int(EventConfig.aColumnWidths[0]);

    // Eventzeit schreiben
    if (WriteEventTime(pEntry     := pEntry,
                       pRoom      := #tmpRoom,
                       sFont      := sFont,
                       sTextColor := sTextColor,
                       sBackColor := sBackColor) = false) then
      bSuccessful := false;
    end_if;
  end_if;

  // Parameter1
  //------------------------------------------------------------
  // Prüfen ob Parameter1 dargestellt werden soll
  if (ColumnChoice AND 2#00010) then

    // Platz für Parameter1 bestimmen
    tmpRoom.xy1.x := tmpRoom.xy2.x;
    tmpRoom.xy2.x := tmpRoom.xy1.x + to_int(EventConfig.aColumnWidths[1]);

    // Parameter1 ausgeben
    if (WriteParameter1(pEntry    := pEntry,
                       pRoom      := #tmpRoom,
                       sFont      := sFont,
                       sTextColor := sTextColor,
                       sBackColor := sBackColor) = false) then
      bSuccessful := false;
    end_if;

  end_if;

  // Alarmnummer schreiben
  //------------------------------------------------------------
  // Prüfen ob Alarmnummer dargestellt werden soll
  if (ColumnChoice AND 2#00100) then

    // Platz für Alarmnummer bestimmen
    tmpRoom.xy1.x := tmpRoom.xy2.x;
    tmpRoom.xy2.x := tmpRoom.xy1.x + to_int(EventConfig.aColumnWidths[2]);

    // Alarmcode ausgeben
    if (WriteAlarmNo(pEntry     := pEntry,
                     pRoom      := #tmpRoom,
                     sFont      := sFont,
                     sTextColor := sTextColor,
                     sBackColor := sBackColor) = false) then
      bSuccessful := false;
    end_if;

  end_if;

  // Parameter2 schreiben
  //------------------------------------------------------------
  // Prüfen ob Parameter2 dargestellt werden soll
  if (ColumnChoice AND 2#01000) then

    // Platz für Parameter2 bestimmen
    tmpRoom.xy1.x := tmpRoom.xy2.x;
    tmpRoom.xy2.x := tmpRoom.xy1.x + to_int(EventConfig.aColumnWidths[3]);

    // Parameter2 ausgeben
    if (WriteParameter2(pEntry     := pEntry,
                        pRoom      := #tmpRoom,
                        sFont      := sFont,
                        sTextColor := sTextColor,
                        sBackColor := sBackColor) = false) then
      bSuccessful := false;
    end_if;

  end_if;

  // Eventtext
  //------------------------------------------------------------
  // Prüfen ob Eventtext dargestellt werden soll
  if (ColumnChoice AND 2#10000) then

    // Platz für Eventtext
    tmpRoom.xy1.x := tmpRoom.xy2.x + Event_TextOffset;
    tmpRoom.xy2.x := tmpRoom.xy1.x + to_int(EventConfig.aColumnWidths[4]);
    if (tmpRoom.xy2.x > (pRoom^.xy2.x)) then
      tmpRoom.xy2.x := pRoom^.xy2.x;
    end_if;

    // Eventtext ausgeben
    if (WriteEventText(pEntry     := pEntry,
                       pRoom      := #tmpRoom,
                       sFont      := sFont,
                       sTextColor := sTextColor,
                       sBackColor := sBackColor) = false) then
      bSuccessful := false;
    end_if;

  end_if;

END_FUNCTION

FUNCTION EventJournal::CalcWidth

  // Breite der Zeile berechnen
  //--------------------------------------------------------------------------------------------

  // Konfiguration der Spalten lesen
  ColumnChoice := ColumnChoice.Read();

  LineWidth := 0;

  // Eventzeit
  if (ColumnChoice AND 2#00001) then
    LineWidth += EventConfig.aColumnWidths[0];
  end_if;

  // Parameter1
  if (ColumnChoice AND 2#00010) then
    LineWidth += EventConfig.aColumnWidths[1];
  end_if;

  // Alarmnummer
  if (ColumnChoice AND 2#00100) then
    LineWidth += EventConfig.aColumnWidths[2];
  end_if;

  // Parameter2
  if (ColumnChoice AND 2#01000) then
    LineWidth += EventConfig.aColumnWidths[3];
  end_if;

  // Beschreibung
  if (ColumnChoice AND 2#10000) then
    LineWidth += EventConfig.aColumnWidths[4];
  end_if;

END_FUNCTION

FUNCTION VIRTUAL GLOBAL EventJournal::DisplayFilter::Write
	VAR_INPUT
		input (EAX) 	: EventJournal::T_BITS;
	END_VAR
	VAR_OUTPUT
		result (EAX) 	: EventJournal::T_BITS;
	END_VAR

  VAR
    mydat : UDINT;
	  para  : UDINT;
  END_VAR

  mydat := DisplayFilter$UDINT;
  para  := input$UDINT;

  if(para and 16#80000000) then
    if(para = 16#80000000) then
	    mydat := mydat or 16#80000000;
	  else
      mydat := mydat or (para and 16#7FFFFFFF);
    end_if;
  else
    if(para = 0) then
      mydat := mydat and 16#7FFFFFFF;
    else
	  mydat := mydat and (16#FFFFFFFF xor para);
	  end_if;
  end_if;

  result        := mydat;
  DisplayFilter := mydat;

END_FUNCTION

FUNCTION EventJournal::ChkEventDispFilter
	VAR_INPUT
		pEventEntry : ^_SINGLEALARM;
	END_VAR
	VAR_OUTPUT
		FilterOK 	: BOOL;
	END_VAR

  FilterOK := FALSE;

  if (pEventEntry <> NIL) then

    if ( ((pEventEntry^.entrytype = Event_SystemCat1)  & (DisplayFilter and 16#0001)) |
         ((pEventEntry^.entrytype = Event_SystemCat2)  & (DisplayFilter and 16#0002)) |
         ((pEventEntry^.entrytype = Event_SystemCat3)  & (DisplayFilter and 16#0004)) |
         ((pEventEntry^.entrytype = Event_SystemCat4)  & (DisplayFilter and 16#0008)) |
         ((pEventEntry^.entrytype = EVENT_ALARM)       & (DisplayFilter and 16#0010)) |

         ((pEventEntry^.entrytype = EVENT_SWITCHOFF)   & (DisplayFilter and 16#0020)) |
         ((pEventEntry^.entrytype = EVENT_SWITCHON)    & (DisplayFilter and 16#0020)) |

         ((pEventEntry^.entrytype = EVENT_USERLOGIN)   & (DisplayFilter and 16#0040)) |
         ((pEventEntry^.entrytype = EVENT_USERLOGOUT)  & (DisplayFilter and 16#0040)) |

         ((pEventEntry^.entrytype = EVENT_MENUCHANGE)  & (DisplayFilter and 16#0080)) |
         ((pEventEntry^.entrytype = EVENT_DATECHANGE)  & (DisplayFilter and 16#0080)) |
         ((pEventEntry^.entrytype = EVENT_VALUECHANGE) & (DisplayFilter and 16#0080)) |
         ((pEventEntry^.entrytype = EVENT_TIMECHANGE)  & (DisplayFilter and 16#0080)) |

         ((pEventEntry^.entrytype = EVENT_USEREVENT)   & (DisplayFilter and 16#0100)) |

         ((pEventEntry^.entrytype = EVENT_OPCHANGE)    & (DisplayFilter and 16#0200)) ) then

      FilterOK := TRUE;

    else

      FilterOK := FALSE;

    end_if;

  end_if;

END_FUNCTION

FUNCTION __CDECL VIRTUAL GLOBAL EventJournal::GetEvent
	VAR_INPUT
		ped 	: ^_EDITOR;
		pe 	: ^_EVENT;
	END_VAR
	VAR_OUTPUT
		retcode (EAX) 	: _DOIT;
	END_VAR
VAR
    doit : BOOL;
	eat : BOOL;
END_VAR

  retcode := _IDLE;

  if(Focus = TRUE) then
    eat := false;
    if(pe^.ftype = _EVENT_KEYPRESS) then
      doit := FALSE;
      case pe^.scancode of
        _UP   : if(Scroll.position.pos > 0) then
                  doit := TRUE;
                end_if;
        _DOWN : if(Scroll.position.pos < (Scroll.position.no - 1)) then
                  doit := TRUE;
                end_if;
        _RIGHT: if(Scroll.hlevel.active = TRUE) then
                  if(Scroll.hposition.pos < (Scroll.hposition.no - 1)) then
//                    Scroll.hposition.pos += (Scroll.out_room.xy2.x - Scroll.out_room.xy1.x) / 4;
                    pe^.scancode := _PGRIGHT;
                    doit := TRUE;
                  end_if;
                end_if;
        _LEFT : if(Scroll.hlevel.active = TRUE) then
                  if(Scroll.hposition.pos > 0) then
//                    Scroll.hposition.pos -= (Scroll.out_room.xy2.x - Scroll.out_room.xy1.x) / 4;
                    pe^.scancode := _PGLEFT;
                    doit := TRUE;
                  end_if;
                end_if;
        _PGLEFT,
        _PGRIGHT,
        _PGUP,
        _PGDOWN : doit := TRUE;
      end_case;
    elsif(pe^.ftype = _EVENT_SHUTTLEDEC) then
      if(Scroll.position.pos > 0) then
        doit := TRUE;
        eat  := TRUE;
      end_if;
    elsif(pe^.ftype = _EVENT_SHUTTLEINC) then
      if(Scroll.position.pos < (Scroll.position.no - 1)) then
        doit := TRUE;
        eat  := TRUE;
      end_if;
    else
      doit := TRUE;
      if((pe^.ftype = _EVENT_HIDMOVE)&(FocusJustGiven = TRUE)) then
        if((pe^.dot.x >= Scroll.out_room.xy1.x)&(pe^.dot.x <= Scroll.out_room.xy2.x)&
           (pe^.dot.y >= Scroll.out_room.xy1.y)&(pe^.dot.y <= Scroll.out_room.xy2.y)) then
          pe^.ftype := _EVENT_HIDPRESS;
          eat       := TRUE;
        end_if;
      end_if;
    end_if;

    FocusJustGiven := FALSE;

    if(doit = TRUE) then

      // --- HubChr 31.05.2016 we don't have a cursor so we don't want to scroll line by line -> set position to first or last visible entry upon scroll event
      if pe^.ftype = _EVENT_HIDPRESS &
        ((pe^.dot.x >= Scroll.level.room.xy1.x) & (pe^.dot.x <= Scroll.level.room.xy2.x)) then // is the x-coord of the press event within the scrollbar?

        if((pe^.dot.y >= Scroll.level.room.xy1.y+(LEVELBUTTON_HEIGHT*Scroll.level.pguppgdown)) & (pe^.dot.y <= Scroll.level.room.xy1.y+LEVELBUTTON_HEIGHT+(LEVELBUTTON_HEIGHT*Scroll.level.pguppgdown))) then // upper scrollbutton
          Scroll.position.pos := scroll.position.begin;
        elsif
          ((pe^.dot.y >= Scroll.level.room.xy2.y-LEVELBUTTON_HEIGHT-(LEVELBUTTON_HEIGHT*Scroll.level.pguppgdown)) & (pe^.dot.y <= scroll.level.room.xy2.y-(LEVELBUTTON_HEIGHT*Scroll.level.pguppgdown))) then // lower scrollbutton
          Scroll.position.pos := Scroll.position.begin + Scroll.position.height-1;
        end_if;
      end_if;
      // --- End HubChr

      Run_SCROLL(#Scroll, pe);

      case(pe^.ftype) of
        _EVENT_KEYPRESS   : eat := TRUE;
        _EVENT_HIDPRESS,
        _EVENT_HIDMOVE,
        _EVENT_HIDRELEASE : if((pe^.dot.x >= Scroll.out_room.xy1.x)&(pe^.dot.x <= Scroll.out_room.xy2.x)&
                               (pe^.dot.y >= Scroll.out_room.xy1.y)&(pe^.dot.y <= Scroll.out_room.xy2.y)) then
                              eat := TRUE;
                            end_if;

      end_case;

      if(eat = TRUE) then
        init_EVENT(pe);     // eat event
        retcode := _IDIDIT;
      end_if;
    end_if;

    ActPos := Scroll.position.pos;
  end_if;

END_FUNCTION

FUNCTION EventJournal::SplitPath
	VAR_OUTPUT
		retcode 	: DINT;
	END_VAR
VAR
	tmpLength : UDINT;
  tmpCounter : USINT;
  i : USINT;
END_VAR

  // ***************************************************************
  // Diese Methode teilt den String mit dem Ordnerpfad in Teile auf,
  // um danach die einzelnen Ordner erstellen zu können.
  // Zum Beispiel: "C:\Hugo\Sepp\Hans", wird aufgeteilt in:
  //    1. Ordnerpfad -> "C:\Hugo"
  //    2. Ordnerpfad -> "C:\Hugo\Sepp"
  //    3. Ordnerpfad -> "C:\Hugo\Sepp\Hans"
  // ***************************************************************

  retcode := 0;

  tmpCounter := 0;

  // Länge des Ordnerpfades holen
  tmpLength := coSigCLib.StrLen(str:=#aFilename[0]);

  if tmpLength <= 0 then
    retcode := -1;
    return;
  end_if;

  for i := 0 to tmpLength - 1 do

    // Schauen ob im Ordnerpfad ein "\" steht
    if aFilename[i] = '\' then

      if tmpCounter = 0 then

      elsif tmpCounter > 0 then

        // Speichern des Ordnerpfades in einer Struktur
        coSigCLib.StrNCpy(dst0:=#FolderPathList.FolderPaths[tmpCounter].FolderPath[0] , src0:=#aFilename[0], count:=i);

      end_if;

      tmpCounter += 1;

      // Kontrollieren ob das Array groß genug ist
      if tmpCounter > (sizeof(FolderPathList.FolderPaths) / sizeof(FolderPathList.FolderPaths[1])) then

        retcode := -2;

        if (IsCon_coSystemLogging = TRUE) then
          coSystemLogging.LogEventText(pChar:="EventJournal::SplitPath(): Array für die Ordnerpfade ist zu klein!");
        end_if;

        return;
      end_if;

    end_if;

    // Letztes Zeichen
    if i = (tmpLength -1) then

      // Letzten Ordnerpfad speichern (ist der einzige wenn nur ein Ordner im Pfad enthalten ist)
      if tmpCounter > 0 then
        coSigCLib.StrCpy(dst0:=#FolderPathList.FolderPaths[tmpCounter].FolderPath[0], src0:=#aFilename[0]);
        FolderPathList.uiFolderNr := tmpCounter;
      end_if;

    end_if;

  end_for;

END_FUNCTION

//*******************************************************************************************************************************
//  Add e new event for external use    V.1.2, KaiAnd
//*******************************************************************************************************************************
FUNCTION __CDECL VIRTUAL GLOBAL EventJournal::AddEntry
	VAR_INPUT
		ptr 	: ^_SINGLEALARM;
	END_VAR
	VAR_OUTPUT
		retcode (AL) 	: BOOL;
	END_VAR
  VAR
	  NiGive	:	CmdStruct;
  	NiGet		:	Results;
    dDate   : DINT;
    dTime   : DINT;
    dValue  : DINT;
pText : ^_CHAR;
  END_VAR

  // share the new event
  if (IsClientConnected(#ccNewEvent)) then

    NiGive.uiCmd    := 11;            // Command
    NiGive.aPara[0] := (ptr)$DINT;    // pointer to original _SINGLEALARM

    // type of the event
    NiGive.aPara[1] := ptr^.entrytype;

    // Date and Time of the event
    GetEventTime(pEntry:=ptr, pRetdDate:=#dDate, pRetdTime:=#dTime);
    NiGive.aPara[2] := dDate;
    NiGive.aPara[3] := dTime;

    // Parameter 1 of the event
    GetParameter1(pEntry:=ptr, pRetDINT:=#dValue);
    NiGive.aPara[4] := dValue;

    // Alarm-No of the Event
    GetAlarmNo(pEntry:=ptr, pRetDINT:=#dValue);
    NiGive.aPara[5] := dValue;

    // Parameter 2 of the event
    GetParameter2(pEntry:=ptr, pRetDINT:=#dValue);
    NiGive.aPara[6] := dValue;

    // Text of the event
pText  := GetEventText(pEntry:=ptr);
    NiGive.aPara[7] := (GetEventText(pEntry:=ptr))$DINT;

    ccNewEvent.NewInst(#NiGive, #NiGet);

  end_if;

  // call the base function
  retcode := _AlarmDisplay::AddEntry(ptr:=ptr);

END_FUNCTION
